(* IEC 61131-3 sources: POMIRTS_lab3/AS/Library/AsHW, 3 files *)

(* ---- AsHW.typ ---- *)
(********************************************************************
 * COPYRIGHT -- Bernecker + Rainer
 ********************************************************************
 * Library: AsHW
 * File: AsHW.typ
 * Author: B+R
 ********************************************************************
 * Data types of library AsHW
 ********************************************************************)

TYPE

END_TYPE

(* ---- AsHW.fun ---- *)
(********************************************************************
 * COPYRIGHT -- Bernecker + Rainer
 ********************************************************************
 * Library: AsHW
 * File: AsHW.fun
 * Author: B+R
 ********************************************************************
 * Functions and function blocks of library AsHW
 ********************************************************************)

FUNCTION_BLOCK HwGetBatteryInfo	(*evaluates a device's battery state; asynchronous execution*)
	VAR_INPUT
	    enable      : BOOL; 	(*enables execution*)
		pDevice	    : UDINT;	(*device name given as a pointer, e.g., "SL0.SS0.HW"*)
		ordinal     : USINT;	(*ordinal number of the hardware element: 1 = battery in the backplane, 2 = battery in the CPU*)
	END_VAR

	VAR
        i_state     : UINT;		(*internal variable*)
        i_result    : UINT;		(*internal variable*)
	END_VAR

	VAR_OUTPUT
		status	    : UINT; 	(*execution status: ERR_OK, ERR_FUB_ENABLE_FALSE, ERR_FUB_BUSY, 0xXXXX = see help*)
		state	    : USINT;	(*battery status: ASHW_BATTERY_LOW, ASHW_BATTERY_OK, ASHW_BATTERY_NOTEST, ASHW_BATTERY_MISSING*)
	END_VAR
END_FUNCTION_BLOCK

FUNCTION_BLOCK HwGetTemperature	(*evaluates the temperature state; asynchronous execution*)
	VAR_INPUT
		enable      : BOOL; 	(*enables execution*)
		pDevice	    : UDINT; 	(*device name given as a pointer, e.g., "SL0.SS0.HW"*)
		ordinal	    : USINT;	(*ordinal number of the hardware element: 1 = cooling plate temperature, 2 = module temperature*)
	END_VAR

	VAR
		i_state     : UINT;		(*internal variable*)
        i_result    : UINT;		(*internal variable*)
	END_VAR

	VAR_OUTPUT
	    status	    : UINT; 	(*execution status: ERR_OK, ERR_FUB_ENABLE_FALSE, ERR_FUB_BUSY, 0xXXXX = see help*)
        temperature : UDINT;	(*temperature [1/10°C]*)
	END_VAR
END_FUNCTION_BLOCK

FUNCTION_BLOCK HwGetMode		(*evaluates the mode switch position; asynchronous execution*)
	VAR_INPUT
		enable      : BOOL; 	(*enables execution*)
		pDevice	    : UDINT; 	(*device name given as a pointer, e.g., "SL0.SS0.HW"*)
		ordinal	    : USINT;	(*ordinal number of the hardware element (default 1)*)
	END_VAR

	VAR
		i_state     : UINT;		(*internal variable*)
        i_result    : UINT;		(*internal variable*)
	END_VAR

	VAR_OUTPUT
		status      : UINT; 	(*execution status: ERR_OK, ERR_FUB_ENABLE_FALSE, ERR_FUB_BUSY, 0xXXXX = see help*)
        mode        : USINT;	(*mode switch*)
	END_VAR

END_FUNCTION_BLOCK

FUNCTION_BLOCK HwGetNode		(*evaluates the node switch position; asynchronous execution*)
	VAR_INPUT
		enable      : BOOL; 	(*enables execution*)
		pDevice	    : UDINT; 	(*device name given as a pointer, e.g., "SL0.SS0.HW"*)
		ordinal	    : USINT;	(*ordinal number of the hardware element (default 1)*)
	END_VAR

	VAR
        i_state     : UINT;		(*internal variable*)
		i_result    : UINT;		(*internal variable*)
        i_reserve   : UDINT;	(*internal variable*)
	END_VAR

	VAR_OUTPUT
		status      : UINT; 	(*execution status: ERR_OK, ERR_FUB_ENABLE_FALSE, ERR_FUB_BUSY, 0xXXXX = see help*)
        node        : USINT;	(*node number (decimal)*)
	END_VAR
END_FUNCTION_BLOCK

FUNCTION_BLOCK HwSetUserLED		(*operates user LEDs; asynchronous execution*)
	VAR_INPUT
		enable      : BOOL; 	(*enables execution*)
		pDevice	    : UDINT; 	(*device name given as a pointer, e.g., "SL0.SS0.HW"*)
		ordinal	    : USINT;	(*ordinal number of the hardware element, e.g., PPx00 -> ordinal = 1*)
		value	    : USINT;	(*1 =  sets user LED (ASHW_USER_LED_ON), 0 =  clears user LED*)
	END_VAR

	VAR
        i_state     : UINT;		(*internal variable*)
        i_result    : UINT;		(*internal variable*)
	END_VAR

	VAR_OUTPUT
		status	    : UINT; 	(*execution status: ERR_OK, ERR_FUB_ENABLE_FALSE, ERR_FUB_BUSY, 0xXXXX = see help*)
	END_VAR
END_FUNCTION_BLOCK

FUNCTION HwSetBeep : UINT		(*operates the internal speaker*)
	VAR_INPUT
		frequency	:UDINT;		(*beep frequency Hz (40 - 15000)*)
		beepTime	:UDINT;		(*beep duration msec (minimum 10msec)*)
	END_VAR
END_FUNCTION

(* ---- AsHW.var ---- *)
(********************************************************************
 * COPYRIGHT -- Bernecker + Rainer
 ********************************************************************
 * Library: AsHW
 * File: AsHW.var
 * Author: B+R
 ********************************************************************
 * Local variables of library AsHW
 ********************************************************************)

VAR CONSTANT
	ERR_ASHW_INVALID_BEEP_PARAMETER	: UINT	:= 28852;	(*invalid beep parameter*)
	ERR_ASHW_INVALID_ORDINAL	: UINT	:= 28851;	(*invalid ordinal number*)
	ERR_ASHW_INVALID_DEVICE	: UINT	:= 28850;		(*invalid device*)
	ASHW_BATTERY_MISSING	: USINT	:= 3;			(*reserved (currently not used)*)
	ASHW_BATTERY_NOTEST	: USINT	:= 2;				(*reserved (currently not used)*)
	ASHW_USER_LED_ON	: USINT	:= 1;				(*user LED on*)
	ASHW_BATTERY_LOW	: USINT	:= 0;				(*battery empty or not present*)
	ASHW_BATTERY_OK	: USINT	:= 1;					(*battery OK*)
END_VAR
